// Mitsubishi GX Works2 project: TARGIL_B   PLC: FX3G

// global labels: Global1
VAR_GLOBAL CONSTANT
  RE_timer : INT := 60;
END_VAR
VAR_GLOBAL
  X_0 AT X000 : BOOL;
  Y_1 AT Y001 : BOOL;
  X_2 AT X002 : BOOL;
  Y_2 AT Y002 : BOOL;
  X_1 AT X001 : BOOL;
  X_7 AT X007 : BOOL;
  TC_timer6 AT TC6 : BOOL;
  X_6 AT X006 : BOOL;
  Y_6 AT Y006 : BOOL;
  TS6 AT TS6 : BOOL;
  TS6_timer AT TS6 : BOOL;
  D_REGISTER AT D1100 : REAL;
END_VAR
VAR_GLOBAL CONSTANT
  VAL : REAL := 6.0;
END_VAR
VAR_GLOBAL
  X_10 AT X010 : BOOL;
  M_11 AT M11 : BOOL;
  M_12 AT M12 : BOOL;
END_VAR

// task Task_01 (event TRUE, interval 0, priority 31): POU_01

PROGRAM POU_01
(* structured ladder/FBD written out as ST: instructions are called as NAME(EN, inputs, outputs); _pN, _eN, _tN stand for wires *)
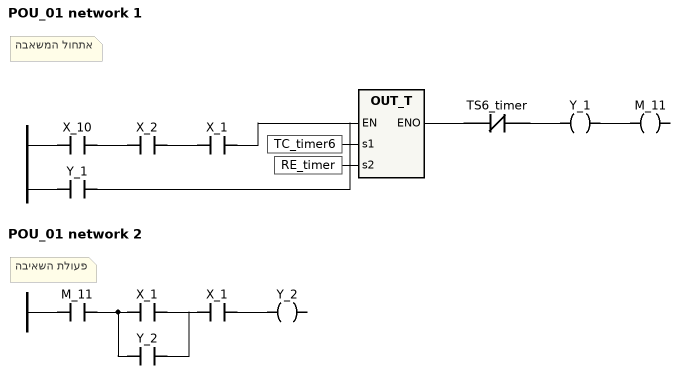
(* network 1 *)
(* אתחול המשאבה *)
_e1 := OUT_T((X_10 AND X_2 AND X_1) OR Y_1, TC_timer6, RE_timer);
_p2 := _e1 AND NOT TS6_timer;
Y_1 := _p2;
M_11 := _p2;
(* network 2 *)
(* פעולת השאיבה *)
Y_2 := ((M_11 AND X_1) OR (M_11 AND Y_2)) AND X_1;
END_PROGRAM
